// TIA Portal V19 export
DATA_BLOCK "A01_Straightener_Ax"   // DB22, Motion_DB
// stored: InstanceOfName TO_PositioningAxis, OfSystemLibElement TO_PositioningAxis, OfSystemLibVersion 8.0
TO_PositioningAxis   // technology object, version 8.0
// stored: Connection Interface Actor, InputAddress 3504, OutputAddress 3504
// stored: Connection Interface Sensor[1], InputAddress 3504, OutputAddress 3504, SensorIndexInActorTelegram 1
// stored: Connection Interface Sensor[2], InputAddress 3504, OutputAddress 3504, SensorIndexInActorTelegram 2
   // // inherited from TO_SpeedAxis
   // // inherited from TO_Axis
   // // inherited from TO_Object
   // VAR
   //    Actor : TO_Struct_Actor;
   //    LoadGear : TO_Struct_LoadGear;
   //    DynamicLimits : TO_Struct_DynamicLimits;
   //    DynamicDefaults : TO_Struct_DynamicDefaults;
   // END_VAR
   // VAR
   //    Position { ExternalWritable := 'False'} : LReal;
   //    ActualPosition { ExternalWritable := 'False'} : LReal;
   //    ActualVelocity { ExternalWritable := 'False'} : LReal;
   //    ActualAcceleration { ExternalWritable := 'False'} : LReal;
   //    OperativeSensor { ExternalWritable := 'False'} : UDInt;
   //    ModuloCycle { ExternalWritable := 'False'} : DInt;
   //    ActualModuloCycle { ExternalWritable := 'False'} : DInt;
   //    Clamping { S7_SetPoint := 'True'} : TO_Struct_Clamping;
   //    Sensor { S7_SetPoint := 'True'} : Array[1..4] of TO_Struct_Sensor;
   //    Extrapolation { S7_SetPoint := 'True'} : TO_Struct_Extrapolation;
   //    Mechanics { S7_SetPoint := 'True'} : TO_Struct_Mechanics;
   //    Properties { ExternalWritable := 'False'; S7_SetPoint := 'True'} : TO_Struct_Properties;
   //    Modulo { S7_SetPoint := 'True'} : TO_Struct_Modulo;
   //    PositionLimits_SW { S7_SetPoint := 'True'} : TO_Struct_PositionLimitsSW;
   //    PositionLimits_HW { S7_SetPoint := 'True'} : TO_Struct_PositionLimitsHW;
   //    Homing { S7_SetPoint := 'True'} : TO_Struct_Homing;
   //    PositionControl { S7_SetPoint := 'True'} : TO_Struct_PositionControl;
   //    TorquePreControl { S7_SetPoint := 'True'} : TO_Struct_TorquePreControl;
   //    SetpointFilter { S7_SetPoint := 'True'} : TO_Struct_SetpointFilter;
   //    DynamicAxisModel { S7_SetPoint := 'True'} : TO_Struct_DynamicAxisModel;
   //    FollowingError { S7_SetPoint := 'True'} : TO_Struct_FollowingError;
   //    CrossPlcSynchronousOperation { S7_SetPoint := 'True'} : TO_Struct_CrossPlcSynchronousOperation;
   //    PositioningMonitoring { S7_SetPoint := 'True'} : TO_Struct_PositioningMonitoring;
   //    StandstillSignal { S7_SetPoint := 'True'} : TO_Struct_StandstillSignal;
   //    StatusPositioning { ExternalWritable := 'False'; S7_SetPoint := 'True'} : TO_Struct_StatusPositioning;
   //    StatusServo { ExternalWritable := 'False'; S7_SetPoint := 'True'} : TO_Struct_StatusServo;
   //    StatusProvidedLeadingValue { ExternalWritable := 'False'; S7_SetPoint := 'True'} : TO_Struct_StatusProvidedLeadingValue;
   //    StatusSensor { ExternalWritable := 'False'; S7_SetPoint := 'True'} : Array[1..4] of TO_Struct_StatusSensor;
   //    StatusExtrapolation { ExternalWritable := 'False'; S7_SetPoint := 'True'} : TO_Struct_StatusExtrapolation;
   //    StatusKinematicsMotion { ExternalWritable := 'False'; S7_SetPoint := 'True'} : TO_Struct_StatusKinematicsMotion;
   // END_VAR
BEGIN
   Actor.DataAdaption := 1;
   Actor.Interface.AddressIn.RID := 16#208072c;
   Actor.Interface.AddressIn.AREA := 16#81;
   Actor.Interface.AddressIn.OFFSET := 3504;
   Actor.Interface.AddressOut.RID := 16#208072d;
   Actor.Interface.AddressOut.AREA := 16#82;
   Actor.Interface.AddressOut.OFFSET := 3504;
   Actor.DriveParameter.ReferenceSpeed := 2200.0;
   Actor.DriveParameter.MaxSpeed := 2200.0;
   Actor.DriveParameter.ReferenceTorque := 52.32;
   LoadGear.Numerator := 76;
   LoadGear.Denominator := 10;
   DynamicLimits.MaxVelocity := 50000.0;
   DynamicLimits.Velocity := 50000.0;
   DynamicLimits.MaxAcceleration := 3000.0;
   DynamicLimits.MaxDeceleration := 3000.0;
   DynamicLimits.MaxJerk := 30000.0;
   DynamicDefaults.Velocity := 6000.0;
   DynamicDefaults.EmergencyDeceleration := 8333.33333333333;
   Sensor[2].Existent := true;
   Sensor[2].MountingMode := 2;
   Sensor[1..2].DataAdaption := 1;
   Sensor[1].ActualVelocityMode := 1;
   Sensor[1..2].Interface.AddressIn.RID := 16#208072c;
   Sensor[1..2].Interface.AddressIn.AREA := 16#81;
   Sensor[1..2].Interface.AddressIn.OFFSET := 3504;
   Sensor[1..2].Interface.AddressOut.RID := 16#208072d;
   Sensor[1..2].Interface.AddressOut.AREA := 16#82;
   Sensor[1..2].Interface.AddressOut.OFFSET := 3504;
   Sensor[2].Interface.Number := 2;
   Sensor[1].Parameter.StepsPerRevolution := 1024;
   Sensor[2].Parameter.StepsPerRevolution := 60000;
   Sensor[2].Parameter.DistancePerRevolution := 500.0;
   Sensor[1].Parameter.ReferenceSpeed := 2200.0;
   Sensor[2].Parameter.ReferenceSpeed := 0.0;
   Sensor[2].Parameter.ReferenceVelocity := 0.0;
   Mechanics.LeadScrew := 251.327412;
   Modulo.Enable := true;
   Modulo.Length := 1000000.0;
   Homing.ApproachVelocity := 6000.0;
   Homing.ReferencingVelocity := 1500.0;
   PositionControl.EnableDSC := true;
   PositionControl.InitialOperativeSensor := 2;
   FollowingError.MinVelocity := 600.0;
   StandstillSignal.VelocityThreshold := 300.0;
   _Units.VelocityUnit := 1524;
   Sensor[2].Existent := True;
   Sensor[2].Interface.Number := 2;
   _Actor.Interface.Telegram := 106;
   _Actor.DataAdaptionOffline := True;
   _Sensor[1].Interface.Telegram := 106;
   _Sensor[1].DataAdaptionOffline := True;
   _Sensor[2].Interface.Telegram := 106;
   _Sensor[2].DataAdaptionOffline := True;
END_DATA_BLOCK
